TYPE T_Ctrl_SIf_FOC_Out :
STRUCT
END_STRUCT
END_TYPE

(* stored: Version 1.1.0.1, ProductVersion 3.1.0.23
   DUT T_Ctrl_SIf_FOC_Out: Id {91c79b87-d334-4452-a561-3b6a384d4bb7} *)
